FUNCTION_BLOCK FB_PowerDelay
VAR_INPUT
	iPowerOnButton: BOOL;
	iServicesOnButton: BOOL; //option
	iPowerOffButton: BOOL;
	iIsStationSelected: BOOL;
	iPowerOnDelay: TIME:=T#3S; //option
END_VAR
VAR_OUTPUT
	qPowerState: BOOL;
	qMotionPowerState:BOOL;
END_VAR
VAR
	timPowerOnDelay: TON;
END_VAR







//theme:zqmIUKoe-q0
VAR // added by the converter: edge detectors and wires of the graphical bodies
    _rt1 : R_TRIG;
END_VAR

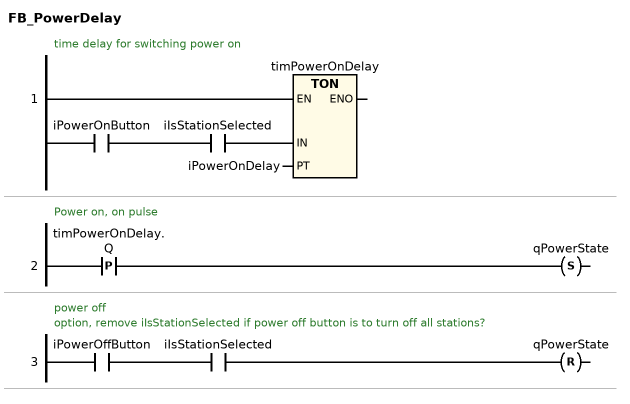
// NETWORK 1
// time delay for switching power on
timPowerOnDelay(IN := iPowerOnButton AND iIsStationSelected, PT := iPowerOnDelay); // TON

// NETWORK 2
// Power on, on pulse
_rt1(CLK := timPowerOnDelay.Q);
qPowerState S= _rt1.Q;

// NETWORK 3
// power off
// option, remove iIsStationSelected if power off button is to turn off all stations?
qPowerState R= iPowerOffButton AND iIsStationSelected;

END_FUNCTION_BLOCK

(* stored: Version 1.1.0.1, ProductVersion 3.1.4024.12
   POU FB_PowerDelay: Id {2b2faf6b-de29-4f2a-aa7d-4834f13ec04e}, SpecialFunc None *)
